TYPE E_ITC_SubsystemControlCode :
(**************************************************************************************
 * 	Application		:	BoxControl Framework
 *	Revision		:	$Revision: 404529 $
 *	Revision date	:	$Date: 2018-04-23 08:21:38 +0200 (Mo., 23 Apr 2018) $
 *	Last changed by	:	$Author: b7bolm $
 *	URL				:	$URL: http://almscdc.swisslog.com/repo/SWPD/Development/BoxControlFramework/20_Release/trunk/01_Software/BCF/BCF/JumpStart/20_Product/10_App/15_Subsystem/10_Lib/10_Conv/01_DUTs/E_ITC_SubSystemControlCode.TcDUT $
 *
 *	Purpose			:	Subsystem control request code
 *
 * ------------------------------------------------------------------------------------
 *	Copyright Swisslog [IP AG], Switzerland. All rights reserved.
 * 
 * ------------------------------------------------------------------------------------
 *	
 * 	Revision History: 
 *
 * 	VERSION			DATE			INITIALS			DESCRIPTION
 *	0.1				01.01.2001		swl					Example
 *
 **************************************************************************************)
(
	NO_CODE							:= 0, // No code
	RESET_ERROR 					:= 1, // Reset Error
	SET_VARIABLE 					:= 5, // Set Variable
	SET_MASTER_SPEED				:= 6, // Set Subsystem master speed
	UPDATE_SYSTEM_TIME				:= 7, // Update system time
	REQUEST_GROUP_POSITION_STATUS	:= 8  // Request status of all groups and positions
);
END_TYPE

(* stored: Version 1.1.0.1, ProductVersion 3.1.4022.12
   DUT E_ITC_SubSystemControlCode: Id {ef168876-a4b7-42d3-af25-8fba33c8de48} *)
